FUNCTION_BLOCK EdgeDetect_VIEW
  (* Version 1.0, 2005-11-13, Goran Cengic, Chalmers *)
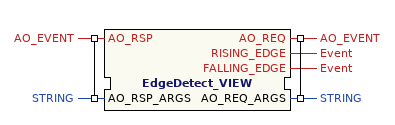
  EVENT_INPUT
    AO_RSP : AO_EVENT WITH AO_RSP_ARGS;
  END_EVENT
  EVENT_OUTPUT
    AO_REQ : AO_EVENT WITH AO_REQ_ARGS;
    RISING_EDGE;
    FALLING_EDGE;
  END_EVENT
  VAR_INPUT
    AO_RSP_ARGS : STRING;
  END_VAR
  VAR_OUTPUT
    AO_REQ_ARGS : STRING;
  END_VAR
END_FUNCTION_BLOCK
